(* IEC 61131-3 sources: brOscatLib/oscatBuild (part 2) *)

(* ---- oscatBuild.fun ---- *)
FUNCTION_BLOCK ACTUATOR_2P (* Actuators *)(* http://www.oscat.de/images/OSCATBuilding/oscat_building100_en.pdf#page=12 *)
    VAR_INPUT
        IN : BYTE;
        TEST : BOOL;
        ARE : BOOL := TRUE;
    END_VAR
    VAR_IN_OUT
        ARX : BOOL;
    END_VAR
    VAR_INPUT
        CYCLE_TIME : TIME;
        SENS : BYTE;
        SELF_ACT_TIME : TIME;
        SELF_ACT_PULSE : TIME;
        SELF_ACT_CYCLES : INT := 1;
    END_VAR
    VAR_OUTPUT
        OUT : BOOL;
        ARO : BOOL;
    END_VAR
    VAR
        timer : AUTORUN;
        pwgen : GEN_PULSE;
    END_VAR
END_FUNCTION_BLOCK
FUNCTION_BLOCK ACTUATOR_3P (* Actuators *)(* http://www.oscat.de/images/OSCATBuilding/oscat_building100_en.pdf#page=13 *)
    VAR_INPUT
        IN : BYTE;
        TEST : BOOL;
        ARE : BOOL := TRUE;
        END_POS : BOOL;
        T_RUN : TIME := TIME#1m0s0ms;
        T_EXT : TIME := TIME#10s0ms;
        T_CAL : TIME := TIME#10m0s0ms;
        T_DIAG : TIME := TIME#14400m0s0ms;
        SWITCH_AVAIL : BOOL;
    END_VAR
    VAR_IN_OUT
        ARX : BOOL;
    END_VAR
    VAR_OUTPUT
        OUT1 : BOOL;
        OUT2 : BOOL;
        POS : BYTE;
        ERROR : BOOL;
        STATUS : BYTE;
    END_VAR
    VAR
        ramp : _RMP_NEXT;
        tx : TIME;
        next_cal : TIME;
        next_diag : TIME;
        last : TIME;
        start : TIME;
    END_VAR
END_FUNCTION_BLOCK
FUNCTION_BLOCK ACTUATOR_A (* Actuators *)(* http://www.oscat.de/images/OSCATBuilding/oscat_building100_en.pdf#page=15 *)
    VAR_INPUT
        I1 : BYTE;
        IS : BOOL;
        I2 : BYTE;
        RV : BOOL;
        DX : BOOL;
        RUNTIME : TIME;
        SELF_ACT_TIME : TIME;
        OUT_MIN : WORD;
        OUT_MAX : WORD;
    END_VAR
    VAR_OUTPUT
        Y : WORD;
    END_VAR
    VAR
        timer : CYCLE_4;
        dx_edge : BOOL;
    END_VAR
END_FUNCTION_BLOCK
FUNCTION_BLOCK ACTUATOR_COIL (* Actuators *)(* http://www.oscat.de/images/OSCATBuilding/oscat_building100_en.pdf#page=16 *)
    VAR_INPUT
        IN : BOOL;
        SELF_ACT_CYCLE : TIME := TIME#14400m0s0ms;
        SELF_ACT_TIME : TIME := TIME#1s0ms;
    END_VAR
    VAR_OUTPUT
        OUT : BOOL;
        STATUS : BYTE;
    END_VAR
    VAR
        last : DWORD;
        init : BOOL;
        tx : DWORD;
        now : DWORD;
    END_VAR
END_FUNCTION_BLOCK
FUNCTION_BLOCK ACTUATOR_PUMP (* Actuators *)(* http://www.oscat.de/images/OSCATBuilding/oscat_building100_en.pdf#page=16 *)
    VAR_INPUT
        IN : BOOL;
        MANUAL : BOOL;
        RST : BOOL;
        MIN_ONTIME : TIME := TIME#10s0ms;
        MIN_OFFTIME : TIME := TIME#10s0ms;
        RUN_EVERY : TIME := TIME#10000m0s0ms;
    END_VAR
    VAR_OUTPUT
        PUMP : BOOL;
    END_VAR
    VAR_IN_OUT
        RUNTIME : UDINT;
        CYCLES : UDINT;
    END_VAR
    VAR
        tx : TIME;
        last_change : TIME;
        meter : ontime;
        old_man : BOOL;
        init : BOOL;
    END_VAR
END_FUNCTION_BLOCK
FUNCTION_BLOCK ACTUATOR_UD (* Actuators *)(* http://www.oscat.de/images/OSCATBuilding/oscat_building100_en.pdf#page=17 *)
    VAR_INPUT
        UD : BOOL;
        ON : BOOL;
        MANUAL : BOOL;
        UP : BOOL;
        DN : BOOL;
        OFF : BOOL;
        YUP_IN : BOOL;
        YDN_IN : BOOL;
        TON : TIME;
        TOFF : TIME;
        OUT_RETURN : BOOL;
    END_VAR
    VAR_OUTPUT
        YUP : BOOL;
        YDN : BOOL;
        STATUS : BYTE;
    END_VAR
    VAR
        tx : TIME;
        last : TIME;
        init : BOOL;
    END_VAR
END_FUNCTION_BLOCK
FUNCTION_BLOCK AUTORUN (* Actuators *)(* http://www.oscat.de/images/OSCATBuilding/oscat_building100_en.pdf#page=19 *)
    VAR_INPUT
        IN : BOOL;
        TEST : BOOL;
        ARE : BOOL := TRUE;
    END_VAR
    VAR_IN_OUT
        ARX : BOOL;
    END_VAR
    VAR_INPUT
        TRUN : TIME;
        TOFF : TIME;
    END_VAR
    VAR_OUTPUT
        OUT : BOOL;
        ARO : BOOL;
    END_VAR
    VAR
        timer : _RMP_B;
        val : BYTE;
    END_VAR
END_FUNCTION_BLOCK
FUNCTION_BLOCK CLICK (* Electrical *)(* http://www.oscat.de/images/OSCATBuilding/oscat_building100_en.pdf#page=47 *)
    VAR_INPUT
        IN : BOOL;
    END_VAR
    VAR_OUTPUT
        Q : BOOL;
        SINGLE : BOOL;
        DOUBLE : BOOL;
        TRIPLE : BOOL;
        STATUS : BYTE;
    END_VAR
    VAR_INPUT
        T_DEBOUNCE : TIME := TIME#10ms;
        T_SHORT : TIME := TIME#200ms;
        T_PAUSE : TIME := TIME#500ms;
        T_RECONFIG : TIME := TIME#1m0s0ms;
    END_VAR
    VAR
        s_in : SW_RECONFIG;
        tx : TIME;
        state : INT;
        last : TIME;
    END_VAR
END_FUNCTION_BLOCK
FUNCTION_BLOCK CLICK_MODE (* Electrical *)(* http://www.oscat.de/images/OSCATBuilding/oscat_building100_en.pdf#page=49 *)
    VAR_INPUT
        IN : BOOL;
    END_VAR
    VAR_OUTPUT
        SINGLE : BOOL;
        DOUBLE : BOOL;
        LONG : BOOL;
        TP_LONG : BOOL;
    END_VAR
    VAR_INPUT
        T_LONG : TIME := TIME#500ms;
    END_VAR
    VAR
        Timer : TP;
        cnt : INT;
        last : BOOL;
    END_VAR
END_FUNCTION_BLOCK
FUNCTION_BLOCK DEBOUNCE (* Electrical *)(* http://www.oscat.de/images/OSCATBuilding/oscat_building100_en.pdf#page=49 *)
    VAR_INPUT
        IN : BOOL;
        TD : TIME;
        PM : BOOL;
    END_VAR
    VAR_OUTPUT
        Q : BOOL;
    END_VAR
    VAR
        deb : TOF;
    END_VAR
END_FUNCTION_BLOCK
FUNCTION_BLOCK DIMM_2 (* Electrical *)(* http://www.oscat.de/images/OSCATBuilding/oscat_building100_en.pdf#page=50 *)
    VAR_INPUT
        SET : BOOL;
        VAL : BYTE := 255;
        I1 : BOOL;
        I2 : BOOL;
        RST : BOOL;
        T_DEBOUNCE : TIME := TIME#10ms;
        T_ON_MAX : TIME := TIME#0ms;
        T_DIMM_START : TIME := TIME#1s0ms;
        T_DIMM : TIME := TIME#3s0ms;
        MIN_ON : BYTE := 50;
        MAX_ON : BYTE := 255;
        RST_OUT : BOOL := TRUE;
        SOFT_DIMM : BOOL := TRUE;
        DBL1_TOG : BOOL;
        DBL2_TOG : BOOL;
        DBL1_SET : BOOL;
        DBL2_SET : BOOL;
        DBL1_POS : BYTE;
        DBL2_POS : BYTE;
    END_VAR
    VAR_OUTPUT
        Q : BOOL := FALSE;
        D1 : BOOL;
        D2 : BOOL;
    END_VAR
    VAR_IN_OUT
        OUT : BYTE;
    END_VAR
    VAR
        t1 : TOF;
        t2 : TOF;
        dc1 : CLICK_MODE;
        dc2 : CLICK_MODE;
        t3 : TON;
        dim : _RMP_B;
    END_VAR
END_FUNCTION_BLOCK
FUNCTION_BLOCK DIMM_I (* Electrical *)(* http://www.oscat.de/images/OSCATBuilding/oscat_building100_en.pdf#page=52 *)
    VAR_INPUT
        SET : BOOL;
        VAL : BYTE := 255;
        IN : BOOL;
        RST : BOOL;
        T_DEBOUNCE : TIME := TIME#10ms;
        T_RECONFIG : TIME := TIME#10s0ms;
        T_ON_MAX : TIME := TIME#0ms;
        T_DIMM_START : TIME := TIME#1s0ms;
        T_DIMM : TIME := TIME#3s0ms;
        MIN_ON : BYTE := 50;
        MAX_ON : BYTE := 255;
        SOFT_DIMM : BOOL := TRUE;
        DBL_TOGGLE : BOOL;
        RST_OUT : BOOL;
    END_VAR
    VAR_OUTPUT
        Q : BOOL := FALSE;
        DBL : BOOL;
    END_VAR
    VAR_IN_OUT
        OUT : BYTE;
    END_VAR
    VAR
        config : SW_RECONFIG;
        decode : CLICK_MODE;
        t3 : TON;
        dim : _RMP_B;
        dir : BOOL;
    END_VAR
END_FUNCTION_BLOCK
FUNCTION_BLOCK F_LAMP (* Electrical *)(* http://www.oscat.de/images/OSCATBuilding/oscat_building100_en.pdf#page=54 *)
    VAR_INPUT
        SWITCH : BOOL;
        DIMM : BYTE := 255;
        RST : BOOL;
    END_VAR
    VAR_OUTPUT
        LAMP : BYTE;
        STATUS : BYTE;
    END_VAR
    VAR_IN_OUT
        ONTIME : UDINT;
        CYCLES : UDINT;
    END_VAR
    VAR_INPUT
        T_NO_DIMM : UINT := 100;
        T_MAINTENANCE : UINT := 15000;
    END_VAR
    VAR
        runtime : ONTIME;
    END_VAR
END_FUNCTION_BLOCK
FUNCTION_BLOCK PULSE_LENGTH (* Electrical *)(* http://www.oscat.de/images/OSCATBuilding/oscat_building100_en.pdf#page=56 *)
    VAR_INPUT
        IN : BOOL;
    END_VAR
    VAR_OUTPUT
        SHORT : BOOL;
        MIDDLE : BOOL;
        LONG : BOOL;
    END_VAR
    VAR_INPUT
        T_SHORT : TIME := TIME#100ms;
        T_LONG : TIME := TIME#1s0ms;
    END_VAR
    VAR
        tx : TIME;
        tn : TIME;
        edge_ : BOOL;
    END_VAR
END_FUNCTION_BLOCK
FUNCTION_BLOCK PULSE_T (* Electrical *)(* http://www.oscat.de/images/OSCATBuilding/oscat_building100_en.pdf#page=56 *)
    VAR_INPUT
        IN : BOOL;
        T1 : TIME;
        T2 : TIME;
        RST : BOOL;
    END_VAR
    VAR_OUTPUT
        Q : BOOL;
    END_VAR
    VAR
        init : BOOL;
        last : TIME;
        tx : TIME;
        edge_ : BOOL;
    END_VAR
END_FUNCTION_BLOCK
FUNCTION_BLOCK SW_RECONFIG (* Electrical *)(* http://www.oscat.de/images/OSCATBuilding/oscat_building100_en.pdf#page=57 *)
    VAR_INPUT
        IN : BOOL;
        TD : TIME;
        TR : TIME;
    END_VAR
    VAR_OUTPUT
        Q : BOOL;
    END_VAR
    VAR
        T1 : TON;
        T2 : TON;
        INV : BOOL;
    END_VAR
END_FUNCTION_BLOCK
FUNCTION_BLOCK SWITCH_I (* Electrical *)(* http://www.oscat.de/images/OSCATBuilding/oscat_building100_en.pdf#page=58 *)
    VAR_INPUT
        SET : BOOL;
        IN : BOOL;
        RST : BOOL;
        T_DEBOUNCE : TIME := TIME#10ms;
        T_RECONFIG : TIME := TIME#1s0ms;
        T_ON_MAX : TIME := TIME#0ms;
    END_VAR
    VAR_OUTPUT
        Q : BOOL;
    END_VAR
    VAR
        state : BYTE;
        edge_ : BOOL;
        r_edge : BOOL;
        T_on : TIME;
        tx : TIME;
    END_VAR
END_FUNCTION_BLOCK
FUNCTION_BLOCK SWITCH_X (* Electrical *)(* http://www.oscat.de/images/OSCATBuilding/oscat_building100_en.pdf#page=59 *)
    VAR_INPUT
        IN1 : BOOL;
        IN2 : BOOL;
        IN3 : BOOL;
        IN4 : BOOL;
        IN5 : BOOL;
        IN6 : BOOL;
    END_VAR
    VAR_OUTPUT
        Q1 : BOOL;
        Q2 : BOOL;
        Q3 : BOOL;
        Q4 : BOOL;
        Q5 : BOOL;
        Q6 : BOOL;
        Q31 : BOOL;
        Q41 : BOOL;
        Q51 : BOOL;
        Q61 : BOOL;
        Q32 : BOOL;
        Q42 : BOOL;
        Q52 : BOOL;
        Q62 : BOOL;
    END_VAR
    VAR_INPUT
        T_DEBOUNCE : TIME := TIME#50ms;
    END_VAR
    VAR
        init : BOOL;
        T1 : TOF;
        T2 : TOF;
        T3 : TOF;
        T4 : TOF;
        T5 : TOF;
        T6 : TOF;
        tx : TIME;
        x1 : BOOL;
        x2 : BOOL;
        E1 : BOOL;
        E2 : BOOL;
    END_VAR
END_FUNCTION_BLOCK
FUNCTION_BLOCK TIMER_1 (* Electrical *)(* http://www.oscat.de/images/OSCATBasic/oscat_basic333_en.pdf#page=60 *)
    VAR_INPUT
        E : BOOL := TRUE;
        DTI : DT;
        START : TOD;
        DURATION : TIME;
        DAY : BYTE := 2#1111111;
    END_VAR
    VAR_OUTPUT
        Q : BOOL;
        STOP : TIME;
    END_VAR
END_FUNCTION_BLOCK
FUNCTION_BLOCK TIMER_2 (* Electrical *)(* http://www.oscat.de/images/OSCATBuilding/oscat_building100_en.pdf#page=60 *)
    VAR_INPUT
        DT_IN : DT;
        START : TOD;
        DURATION : TIME;
        MODE : BYTE;
        HOLIDAY : BOOL;
    END_VAR
    VAR_OUTPUT
        Q : BOOL;
    END_VAR
    VAR
        last_check : TIME;
        dat : DATE;
        daytime : TOD;
        activation : TIME;
        tx : TIME;
        enabled : BOOL;
        init : BOOL;
        wday : INT;
    END_VAR
    VAR RETAIN
        run_date : DATE;
    END_VAR
END_FUNCTION_BLOCK
FUNCTION TIMER_EVENT_DECODE : BOOL (* Electrical *)(* http://www.oscat.de/images/OSCATBuilding/oscat_building100_en.pdf#page=62 *)
    VAR_INPUT
        EVENT : STRING[STRING_LENGTH];
        LANG : INT;
    END_VAR
    VAR
        pos : INT;
        start : INT;
        stop : INT;
        pt : REFERENCE TO ARRAY[1..255] OF BYTE;
        step : INT;
        tmp : STRING[60];
    END_VAR
    VAR_IN_OUT
        RETVAL : TIMER_EVENT; (*Return value of the function*)
    END_VAR
END_FUNCTION
FUNCTION_BLOCK TIMER_EXT (* Electrical *)(* http://www.oscat.de/images/OSCATBuilding/oscat_building100_en.pdf#page=63 *)
    VAR_INPUT
        ENA : BOOL := TRUE;
        ON : BOOL;
        OFF : BOOL;
        MAN : BOOL;
        SWITCH : BOOL;
        DT_IN : DT;
        SUN_RISE : TOD;
        SUN_SET : TOD;
        HOLIDAY : BOOL;
        T_DEBOUNCE : TIME := TIME#100ms;
        T_RISE_START : TIME;
        T_RISE_STOP : TIME;
        T_SET_START : TIME;
        T_SET_STOP : TIME;
        T_DAY_START : TOD;
        T_DAY_STOP : TOD;
        ENABLE_SATURDAY : BOOL;
        ENABLE_SUNDAY : BOOL;
        ENABLE_HOLIDAY : BOOL;
    END_VAR
    VAR_OUTPUT
        Q : BOOL;
        STATUS : BYTE;
    END_VAR
    VAR
        mx : MANUAL_2;
        deb : DEBOUNCE;
        tdx : TOD;
        wdx : INT;
        tc : TIME;
        tx : DWORD;
        tl : DWORD;
        qx : BOOL;
        init : BOOL;
    END_VAR
END_FUNCTION_BLOCK
FUNCTION_BLOCK TIMER_P4 (* Electrical *)(* http://www.oscat.de/images/OSCATBuilding/oscat_building100_en.pdf#page=65 *)
    VAR_INPUT
        DTIME : DT;
        TREF_0 : TOD;
        TREF_1 : TOD;
        HOLY : BOOL;
        L0 : BOOL;
        L1 : BOOL;
        L2 : BOOL;
        L3 : BOOL;
        OFS : BYTE;
        ENQ : BOOL;
        MAN : BOOL;
        MI : BYTE;
        RST : BOOL;
    END_VAR
    VAR_IN_OUT
        PROG : ARRAY[0..array_max] OF TIMER_EVENT;
    END_VAR
    VAR_OUTPUT
        Q0 : BOOL;
        Q1 : BOOL;
        Q2 : BOOL;
        Q3 : BOOL;
        STATUS : BYTE;
    END_VAR
    VAR CONSTANT
        array_max : INT := 63;
        channel_max : INT := 3;
    END_VAR
    VAR
        day_start : DT;
        start : DT;
        event : TIMER_EVENT;
        pos : INT;
        last_execute : DT;
        current_day : DINT;
        mask : BYTE;
        ma : ARRAY[0..channel_max] OF BYTE;
        mo : ARRAY[0..channel_max] OF BYTE;
        qn : ARRAY[0..channel_max] OF BOOL;
        qs : ARRAY[0..channel_max] OF BOOL;
        channel : INT;
        tx : TOD;
    END_VAR
END_FUNCTION_BLOCK
FUNCTION AIR_DENSITY : REAL (* HLK *)(* http://www.oscat.de/images/OSCATBasic/oscat_basic333_en.pdf#page=426 *)
    VAR_INPUT
        T : REAL;
        P : REAL;
        RH : REAL;
    END_VAR
    VAR CONSTANT
        RL : REAL := 287.05;
        RX : REAL := 0.003773319;
    END_VAR
END_FUNCTION
FUNCTION AIR_ENTHALPY : REAL (* HLK *)(* http://www.oscat.de/images/OSCATBasic/oscat_basic333_en.pdf#page=427 *)
    VAR_INPUT
        T : REAL;
        RH : REAL;
    END_VAR
    VAR CONSTANT
        CPL : REAL := 1.00482;
        CW : REAL := 1.86;
        LH : REAL := 2500.78;
    END_VAR
END_FUNCTION
FUNCTION_BLOCK BOILER (* HLK *)(* http://www.oscat.de/images/OSCATBasic/oscat_basic333_en.pdf#page=428 *)
    VAR_INPUT
        T_UPPER : REAL;
        T_LOWER : REAL;
        PRESSURE : BOOL := TRUE;
        ENABLE : BOOL := TRUE;
        REQ_1 : BOOL;
        REQ_2 : BOOL;
        BOOST : BOOL;
        T_UPPER_MIN : REAL := 50;
        T_UPPER_MAX : REAL := 60;
        T_LOWER_ENABLE : BOOL;
        T_LOWER_MAX : REAL := 60;
        T_REQUEST_1 : REAL := 70;
        T_REQUEST_2 : REAL := 50;
        T_REQUEST_HYS : REAL := 5;
        T_PROTECT_HIGH : REAL := 80;
        T_PROTECT_LOW : REAL := 10;
    END_VAR
    VAR_OUTPUT
        HEAT : BOOL;
        ERROR : BOOL;
        STATUS : BYTE;
    END_VAR
    VAR
        edge_ : BOOL;
        boost_mode : BOOL;
        flag_0 : BOOL;
        flag_1 : BOOL;
        flag_2 : BOOL;
    END_VAR
END_FUNCTION_BLOCK
FUNCTION_BLOCK BURNER (* HLK *)(* http://www.oscat.de/images/OSCATBasic/oscat_basic333_en.pdf#page=430 *)
    VAR_INPUT
        IN : BOOL;
        STAGE2 : BOOL;
        OVER_TEMP : BOOL;
        OIL_TEMP : BOOL := TRUE;
        FLAME : BOOL;
        RST : BOOL;
        RST_TIMER : BOOL;
        PRE_HEAT_TIME : TIME := TIME#5s0ms;
        PRE_VENT_TIME : TIME := TIME#15s0ms;
        PRE_IGNITE_TIME : TIME := TIME#5s0ms;
        POST_IGNITE_TIME : TIME := TIME#25s0ms;
        STAGE2_DELAY : TIME := TIME#10s0ms;
        SAFETY_TIME : TIME := TIME#5s0ms;
        LOCKOUT_TIME : TIME := TIME#10s0ms;
        MULTIPLE_IGNITION : BOOL := TRUE;
        KW1 : REAL;
        KW2 : REAL;
    END_VAR
    VAR_OUTPUT
        MOTOR : BOOL;
        COIL1 : BOOL;
        COIL2 : BOOL;
        PRE_HEAT : BOOL;
        IGNITE : BOOL;
        KWH : REAL;
        STATUS : BYTE;
        FAIL : BOOL;
    END_VAR
    VAR_IN_OUT
        RUNTIME1 : UDINT;
        RUNTIME2 : UDINT;
        CYCLES : UDINT;
    END_VAR
    VAR
        state : BYTE;
        last : TIME;
        tx : TIME;
        last_change : TIME;
        timer1 : ONTIME;
        timer2 : ONTIME;
        oil_temp_last : BOOL;
        cycles2 : UDINT;
    END_VAR
END_FUNCTION_BLOCK
FUNCTION DEW_CON : REAL (* HLK *)(* http://www.oscat.de/images/OSCATBasic/oscat_basic333_en.pdf#page=434 *)
    VAR_INPUT
        RH : REAL;
        T : REAL;
    END_VAR
END_FUNCTION
FUNCTION DEW_RH : REAL (* HLK *)(* http://www.oscat.de/images/OSCATBasic/oscat_basic333_en.pdf#page=435 *)
    VAR_INPUT
        VC : REAL;
        T : REAL;
    END_VAR
END_FUNCTION
FUNCTION DEW_TEMP : REAL (* HLK *)(* http://www.oscat.de/images/OSCATBasic/oscat_basic333_en.pdf#page=436 *)
    VAR_INPUT
        RH : REAL;
        T : REAL;
    END_VAR
    VAR CONSTANT
        a : REAL := 7.5;
        b : REAL := 237.3;
    END_VAR
    VAR
        V : REAL;
    END_VAR
END_FUNCTION
FUNCTION HEAT_INDEX : REAL (* HLK *)(* http://www.oscat.de/images/OSCATBasic/oscat_basic333_en.pdf#page=436 *)
    VAR_INPUT
        T : REAL;
        RH : REAL;
    END_VAR
    VAR
        RH2 : REAL;
        T2 : REAL;
    END_VAR
END_FUNCTION
FUNCTION_BLOCK HEAT_METER (* HLK *)(* http://www.oscat.de/images/OSCATBasic/oscat_basic333_en.pdf#page=436 *)
    VAR_INPUT
        TF : REAL;
        TR : REAL;
        LPH : REAL;
        E : BOOL;
        RST : BOOL;
        CP : REAL;
        DENSITY : REAL;
        CONTENT : REAL;
        PULSE_MODE : BOOL;
        RETURN_METER : BOOL;
        AVG_TIME : TIME := TIME#5s0ms;
    END_VAR
    VAR_OUTPUT
        C : REAL;
    END_VAR
    VAR_IN_OUT
        Y : REAL;
    END_VAR
    VAR
        tx : DWORD;
        last : DWORD;
        int1 : FT_INT2;
        edge_ : BOOL;
        x : REAL;
        init : BOOL;
        y_last : REAL;
    END_VAR
END_FUNCTION_BLOCK
FUNCTION_BLOCK HEAT_TEMP (* HLK *)(* http://www.oscat.de/images/OSCATBasic/oscat_basic333_en.pdf#page=33 *)
    VAR_INPUT
        T_EXT : REAL;
        T_INT : REAL;
        OFFSET : REAL;
        T_REQ : REAL;
        TY_MAX : REAL := 70;
        TY_MIN : REAL := 25;
        TY_CONFIG : REAL := 70;
        T_INT_CONFIG : REAL := 20;
        T_EXT_CONFIG : REAL := -15;
        T_DIFF : REAL := 10;
        C : REAL := 1.33;
        H : REAL := 3;
    END_VAR
    VAR_OUTPUT
        TY : REAL;
        HEAT : BOOL;
    END_VAR
    VAR
        tr : REAL;
        tx : REAL;
    END_VAR
END_FUNCTION_BLOCK
FUNCTION_BLOCK LEGIONELLA (* HLK *)(* http://www.oscat.de/images/OSCATBasic/oscat_basic333_en.pdf#page=443 *)
    VAR_INPUT
        MANUAL : BOOL;
        TEMP_BOILER : REAL;
        TEMP_RETURN : REAL := 100;
        DT_IN : DT;
        RST : BOOL;
        T_START : TOD := TIME_OF_DAY#3:0;
        DAY : INT := 7;
        TEMP_SET : REAL := 70;
        TEMP_OFFSET : REAL := 10;
        TEMP_HYS : REAL := 5;
        T_MAX_HEAT : TIME := TIME#10m0s0ms;
        T_MAX_RET : TIME := TIME#10m0s0ms;
        TP_0 : TIME := TIME#5m0s0ms;
        TP_1 : TIME := TIME#5m0s0ms;
        TP_2 : TIME := TIME#5m0s0ms;
        TP_3 : TIME := TIME#5m0s0ms;
        TP_4 : TIME := TIME#5m0s0ms;
        TP_5 : TIME := TIME#5m0s0ms;
        TP_6 : TIME := TIME#5m0s0ms;
        TP_7 : TIME := TIME#5m0s0ms;
    END_VAR
    VAR_OUTPUT
        HEAT : BOOL;
        PUMP : BOOL;
        VALVE0 : BOOL;
        VALVE1 : BOOL;
        VALVE2 : BOOL;
        VALVE3 : BOOL;
        VALVE4 : BOOL;
        VALVE5 : BOOL;
        VALVE6 : BOOL;
        VALVE7 : BOOL;
        RUN : BOOL;
        STATUS : BYTE;
    END_VAR
    VAR
        X1 : TIMER_1;
        x2 : SEQUENCE_8;
        x3 : HYST_1;
        init : BOOL;
    END_VAR
END_FUNCTION_BLOCK
FUNCTION SDD : REAL (* HLK *)(* http://www.oscat.de/images/OSCATBasic/oscat_basic333_en.pdf#page=445 *)
    VAR_INPUT
        T : REAL;
        ICE : BOOL;
    END_VAR
END_FUNCTION
FUNCTION SDD_NH3 : REAL (* HLK *)(* http://www.oscat.de/images/OSCATBasic/oscat_basic333_en.pdf#page=446 *)
    VAR_INPUT
        T : REAL;
    END_VAR
END_FUNCTION
FUNCTION SDT_NH3 : REAL (* HLK *)(* http://www.oscat.de/images/OSCATBasic/oscat_basic333_en.pdf#page=446 *)
    VAR_INPUT
        P : REAL;
    END_VAR
END_FUNCTION
FUNCTION_BLOCK T_AVG24 (* HLK *)(* http://www.oscat.de/images/OSCATBasic/oscat_basic333_en.pdf#page=446 *)
    VAR_INPUT
        TS : INT;
        DTI : DT;
        RST : BOOL;
        T_FILTER : TIME := TIME#10m0s0ms;
        SCALE : REAL := 1;
        OFS : REAL;
    END_VAR
    VAR_OUTPUT
        TA : REAL;
        TP : BOOL;
    END_VAR
    VAR_IN_OUT
        T24 : REAL;
        T24_MAX : REAL;
        T24_MIN : REAL;
    END_VAR
    VAR
        samples : ARRAY[0..47] OF INT;
        pos : INT;
        init : BOOL;
        ft1 : FILTER_I;
        sum : DINT;
        last : DT;
    END_VAR
    VAR
        tmp_max : INT;
        tmp_min : INT;
        i : INT;
    END_VAR
END_FUNCTION_BLOCK
FUNCTION_BLOCK TANK_LEVEL (* HLK *)(* http://www.oscat.de/images/OSCATBuilding/oscat_building100_en.pdf#page=41 *)
    VAR_INPUT
        LEVEL : BOOL;
        LEAK : BOOL;
        ACLR : BOOL;
        MAX_VALVE_TIME : TIME;
        LEVEL_DELAY_TIME : TIME;
    END_VAR
    VAR_OUTPUT
        VALVE : BOOL;
        ALARM : BOOL;
        STATUS : BYTE;
    END_VAR
    VAR
        cx : ACTUATOR_COIL;
        tn : TON;
        tl : TONOF;
        open : BOOL;
    END_VAR
END_FUNCTION_BLOCK
FUNCTION TANK_VOL1 : REAL (* HLK *)(* http://www.oscat.de/images/OSCATBasic/oscat_basic333_en.pdf#page=448 *)
    VAR_INPUT
        TR : REAL;
        TL : REAL;
        H : REAL;
    END_VAR
END_FUNCTION
FUNCTION TANK_VOL2 : REAL (* HLK *)(* http://www.oscat.de/images/OSCATBasic/oscat_basic333_en.pdf#page=448 *)
    VAR_INPUT
        TR : REAL;
        H : REAL;
    END_VAR
END_FUNCTION
FUNCTION_BLOCK TEMP_EXT (* HLK *)(* http://www.oscat.de/images/OSCATBasic/oscat_basic333_en.pdf#page=449 *)
    VAR_INPUT
        T_EXT1 : REAL;
        T_EXT2 : REAL;
        T_EXT3 : REAL;
        T_EXT_CONFIG : BYTE;
        DT_IN : DT;
        T_EXT_MIN : REAL := -40;
        T_EXT_MAX : REAL := 60;
        T_EXT_DEFAULT : REAL := -10;
        HEAT_PERIOD_START : DATE := DATE#1970-9-1;
        HEAT_PERIOD_STOP : DATE := DATE#1970-4-30;
        COOL_PERIOD_START : DATE := DATE#1970-4-1;
        COOL_PERIOD_STOP : DATE := DATE#1970-9-30;
        HEAT_START_TEMP_DAY : REAL := 15;
        HEAT_START_TEMP_NIGHT : REAL := 10;
        HEAT_STOP_TEMP : REAL := 18;
        COOL_START_TEMP_DAY : REAL := 26;
        COOL_START_TEMP_NIGHT : REAL := 26;
        COOL_STOP_TEMP : REAL := 24;
        START_DAY : TOD := TIME_OF_DAY#9:0;
        START_NIGHT : TOD := TIME_OF_DAY#21:0;
        CYCLE_TIME : TIME := TIME#10m0s0ms;
    END_VAR
    VAR_OUTPUT
        T_EXT : REAL;
        HEAT : BOOL;
        COOL : BOOL;
    END_VAR
    VAR
        tx : TIME;
        last_run : TIME;
        init : BOOL;
        cool_start : DATE;
        cool_stop : DATE;
        heat_start : DATE;
        heat_stop : DATE;
        xdate : DATE;
        day : BOOL;
    END_VAR
END_FUNCTION_BLOCK
FUNCTION WATER_CP : REAL (* HLK *)(* http://www.oscat.de/images/OSCATBasic/oscat_basic333_en.pdf#page=452 *)
    VAR_INPUT
        T : REAL;
    END_VAR
    VAR
        Pts : INT := 10;
        data : ARRAY[1..20, 0..1] OF REAL := [0, 4.228, 5, 4.2, 10, 4.188, 15, 4.184, 50, 4.181, 60, 4.183, 70, 4.187, 80, 4.194, 90, 4.204, 100, 4.22];
    END_VAR
END_FUNCTION
FUNCTION WATER_DENSITY : REAL (* HLK *)(* http://www.oscat.de/images/OSCATBasic/oscat_basic333_en.pdf#page=452 *)
    VAR_INPUT
        T : REAL;
        SAT : BOOL;
    END_VAR
    VAR CONSTANT
        a0 : REAL := 999.83952;
        a1 : REAL := 16.952577;
        a2 : REAL := -0.0079905127;
        a3 : REAL := -4.6241757E-05;
        a4 : REAL := 1.0584601E-07;
        a5 : REAL := -2.8103006E-10;
        b : REAL := 0.0168872;
    END_VAR
    VAR
        T2 : REAL;
        T4 : REAL;
    END_VAR
END_FUNCTION
FUNCTION WATER_ENTHALPY : REAL (* HLK *)(* http://www.oscat.de/images/OSCATBasic/oscat_basic333_en.pdf#page=453 *)
    VAR_INPUT
        T : REAL;
    END_VAR
    VAR
        Pts : INT := 11;
        data : ARRAY[1..20, 0..1] OF REAL := [0, 0.06, 10, 42.1, 20, 83.9, 30, 125.8, 40, 167.58, 50, 209.4, 60, 251.2, 70, 293.1, 80, 335, 90, 377, 100, 419.1];
    END_VAR
END_FUNCTION
FUNCTION WCT : REAL (* HLK *)(* http://www.oscat.de/images/OSCATBasic/oscat_basic333_en.pdf#page=453 *)
    VAR_INPUT
        T : REAL;
        V : REAL;
    END_VAR
END_FUNCTION
FUNCTION_BLOCK BLIND_ACTUATOR (* Jalousie *)(* http://www.oscat.de/images/OSCATBuilding/oscat_building100_en.pdf#page=74 *)
    VAR_INPUT
        UP : BOOL;
        DN : BOOL;
        S_IN : BYTE;
        T_UD : TIME := TIME#10s0ms;
        T_ANGLE : TIME := TIME#3s0ms;
        T_LOCKOUT : TIME := TIME#100ms;
    END_VAR
    VAR_OUTPUT
        POS : BYTE;
        ANG : BYTE;
        QU : BOOL;
        QD : BOOL;
        STATUS : BYTE;
    END_VAR
    VAR
        position : RMP_B;
        angle : RMP_B;
        lock : INTERLOCK;
    END_VAR
END_FUNCTION_BLOCK
FUNCTION_BLOCK BLIND_CONTROL (* Jalousie *)(* http://www.oscat.de/images/OSCATBuilding/oscat_building100_en.pdf#page=75 *)
    VAR_INPUT
        UP : BOOL;
        DN : BOOL;
        S_IN : BYTE;
        PI : BYTE;
        AI : BYTE;
        T_UD : TIME;
        T_ANGLE : TIME;
        SENS : BYTE := 5;
        T_LOCKOUT : TIME := TIME#100ms;
    END_VAR
    VAR_OUTPUT
        POS : BYTE;
        ANG : BYTE;
        MU : BOOL;
        MD : BOOL;
        STATUS : BYTE;
    END_VAR
    VAR
        act : BLIND_ACTUATOR;
        delta : BYTE;
        bTimeTest : BOOL := FALSE;
        iPos : BYTE;
        iAngel : BYTE;
    END_VAR
END_FUNCTION_BLOCK
FUNCTION_BLOCK BLIND_CONTROL_S (* Jalousie *)(* http://www.oscat.de/images/OSCATBuilding/oscat_building100_en.pdf#page=78 *)
    VAR_INPUT
        UP : BOOL;
        DN : BOOL;
        S_IN : BYTE := 125;
        PI : BYTE;
        T_UP : TIME;
        T_DN : TIME;
        RU : BOOL;
        RD : BOOL;
        T_LOCKOUT : TIME := TIME#100ms;
        T_EXT : TIME;
        EXT_TRIG : BYTE := 5;
        R_POS_TOP : BYTE := 255;
        R_POS_BOT : BYTE;
    END_VAR
    VAR_OUTPUT
        POS : BYTE;
        MU : BOOL;
        MD : BOOL;
        STATUS : BYTE;
    END_VAR
    VAR
        rmp : _RMP_NEXT;
        tx : TIME;
        last : TIME;
        PI_last : BYTE;
    END_VAR
END_FUNCTION_BLOCK
FUNCTION_BLOCK BLIND_INPUT (* Jalousie *)(* http://www.oscat.de/images/OSCATBuilding/oscat_building100_en.pdf#page=80 *)
    VAR_INPUT
        POS : BYTE;
        ANG : BYTE;
        S1 : BOOL;
        S2 : BOOL;
        IN : BOOL;
        PI : BYTE;
        AI : BYTE;
        SINGLE_SWITCH : BOOL;
        CLICK_EN : BOOL := TRUE;
        CLICK_TIME : TIME := TIME#500ms;
        MAX_RUNTIME : TIME := TIME#1m0s0ms;
        MANUAL_TIMEOUT : TIME := TIME#60m0s0ms;
        DEBOUNCE_TIME : TIME := TIME#20ms;
        DBL_CLK1 : BOOL := FALSE;
        DBL_POS1 : BYTE;
        DBL_ANG1 : BYTE;
        DBL_CLK2 : BOOL := FALSE;
        DBL_POS2 : BYTE := 255;
        DBL_ANG2 : BYTE := 255;
        D1_TOGGLE : BOOL := TRUE;
        D2_TOGGLE : BOOL := TRUE;
        MASTER_MODE : BOOL;
    END_VAR
    VAR_OUTPUT
        QU : BOOL := TRUE;
        QD : BOOL := TRUE;
        STATUS : BYTE;
        PO : BYTE := 255;
        AO : BYTE := 255;
        D1 : BOOL;
        D2 : BOOL;
    END_VAR
    VAR
        s1e : TOF;
        s2e : TOF;
        s1d : CLICK_MODE;
        s2d : CLICK_MODE;
        dir : BOOL;
        tx : TIME;
        last : TIME;
    END_VAR
END_FUNCTION_BLOCK
FUNCTION_BLOCK BLIND_NIGHT (* Jalousie *)(* http://www.oscat.de/images/OSCATBuilding/oscat_building100_en.pdf#page=84 *)
    VAR_INPUT
        UP : BOOL;
        DN : BOOL;
        S_IN : BYTE;
        PI : BYTE;
        AI : BYTE;
        E_NIGHT : BOOL := TRUE;
        E_DAY : BOOL := TRUE;
        DTIN : DT;
        SUNRISE : TOD;
        SUNSET : TOD;
        SUNRISE_OFFSET : TIME;
        SUNSET_OFFSET : TIME;
        NIGHT_POSITION : BYTE;
        NIGHT_ANGLE : BYTE;
    END_VAR
    VAR_OUTPUT
        QU : BOOL;
        QD : BOOL;
        STATUS : BYTE;
        PO : BYTE;
        AO : BYTE;
    END_VAR
    VAR
        night : BOOL;
        last_night : DATE;
        last_day : DATE;
    END_VAR
END_FUNCTION_BLOCK
FUNCTION_BLOCK BLIND_SCENE (* Jalousie *)(* http://www.oscat.de/images/OSCATBuilding/oscat_building100_en.pdf#page=87 *)
    VAR_INPUT
        UP : BOOL;
        DN : BOOL;
        S_IN : BYTE;
        PI : BYTE;
        AI : BYTE;
        ENABLE : BOOL;
        SWRITE : BOOL;
        SCENE : BYTE;
    END_VAR
    VAR_OUTPUT
        QU : BOOL;
        QD : BOOL;
        STATUS : BYTE;
        PO : BYTE;
        AO : BYTE;
    END_VAR
    VAR RETAIN
        sx : ARRAY[0..15, 0..2] OF BYTE;
    END_VAR
    VAR
        x : BYTE;
    END_VAR
END_FUNCTION_BLOCK
FUNCTION_BLOCK BLIND_SECURITY (* Jalousie *)(* http://www.oscat.de/images/OSCATBuilding/oscat_building100_en.pdf#page=89 *)
    VAR_INPUT
        UP : BOOL;
        DN : BOOL;
        S_IN : BYTE;
        PI : BYTE;
        AI : BYTE;
        FIRE : BOOL;
        WIND : BOOL;
        ALARM : BOOL;
        DOOR : BOOL;
        RAIN : BOOL;
        ALARM_UP : BOOL := TRUE;
        WIND_UP : BOOL := TRUE;
        RAIN_UP : BOOL := FALSE;
    END_VAR
    VAR_OUTPUT
        QU : BOOL;
        QD : BOOL;
        STATUS : BYTE;
        PO : BYTE;
        AO : BYTE;
    END_VAR
END_FUNCTION_BLOCK
FUNCTION_BLOCK BLIND_SET (* Jalousie *)(* http://www.oscat.de/images/OSCATBuilding/oscat_building100_en.pdf#page=91 *)
    VAR_INPUT
        UP : BOOL;
        DN : BOOL;
        S_IN : BYTE;
        PI : BYTE;
        AI : BYTE;
        IN : BOOL;
        PX : BYTE;
        AX : BYTE;
        OVERRIDE_MANUAL : BOOL;
        RESTORE_POSITION : BOOL;
        RESTORE_TIME : TIME := TIME#1m0s0ms;
    END_VAR
    VAR_OUTPUT
        QU : BOOL;
        QD : BOOL;
        STATUS : BYTE;
        PO : BYTE;
        AO : BYTE;
    END_VAR
    VAR
        tx : TIME;
        ps : BYTE;
        as : BYTE;
        last : TIME;
    END_VAR
END_FUNCTION_BLOCK
FUNCTION_BLOCK BLIND_SHADE (* Jalousie *)(* http://www.oscat.de/images/OSCATBuilding/oscat_building100_en.pdf#page=93 *)
    VAR_INPUT
        UP : BOOL;
        DN : BOOL;
        S_IN : BYTE;
        PI : BYTE;
        AI : BYTE;
        ENABLE : BOOL;
        SUN : BOOL;
    END_VAR
    VAR_IN_OUT
        CX : CALENDAR;
    END_VAR
    VAR_INPUT
        SUNRISE_OFFSET : TIME := TIME#60m0s0ms;
        SUNSET_PRESET : TIME := TIME#60m0s0ms;
        DIRECTION : REAL := 180;
        ANGLE_OFFSET : REAL := 80;
        SLAT_WIDTH : REAL := 80;
        SLAT_SPACING : REAL := 60;
        SHADE_DELAY : TIME := TIME#1m0s0ms;
        SHADE_POS : BYTE;
    END_VAR
    VAR_OUTPUT
        QU : BOOL;
        QD : BOOL;
        STATUS : BYTE;
        PO : BYTE;
        AO : BYTE;
    END_VAR
    VAR
        angle : REAL;
        sun_delay : TOF;
    END_VAR
END_FUNCTION_BLOCK
FUNCTION_BLOCK BLIND_SHADE_S (* Jalousie *)(* http://www.oscat.de/images/OSCATBuilding/oscat_building100_en.pdf#page=96 *)
    VAR_INPUT
        UP : BOOL;
        DN : BOOL;
        S_IN : BYTE;
        PI : BYTE;
        ENABLE : BOOL;
        SUN : BOOL;
        HORZ1 : REAL := 100;
        HORZ2 : REAL := 260;
        VERT : REAL := 90;
        ALERT : BOOL := FALSE;
    END_VAR
    VAR_IN_OUT
        CX : calendar;
    END_VAR
    VAR_INPUT
        SUNRISE_OFFSET : TIME := TIME#60m0s0ms;
        SUNSET_PRESET : TIME := TIME#60m0s0ms;
        SHADE_DELAY : TIME := TIME#1m0s0ms;
        SHADE_POS : BYTE;
    END_VAR
    VAR_OUTPUT
        QU : BOOL;
        QD : BOOL;
        STATUS : BYTE;
        PO : BYTE;
    END_VAR
    VAR
        sun_delay : TOF;
    END_VAR
END_FUNCTION_BLOCK
FUNCTION BUILDING_VERSION : DWORD (* Other *)(* http://www.oscat.de/images/OSCATBuilding/oscat_building100_en.pdf#page=11 *)
    VAR_INPUT
        IN : BOOL;
    END_VAR
END_FUNCTION

(* ---- PULSE_LENGTH.st ---- *)
FUNCTION_BLOCK PULSE_LENGTH
    (*http://www.oscat.de/images/OSCATBuilding/oscat_building100_en.pdf#page=56*)
    (* read system time *)
    tx := DWORD_TO_TIME(T_PLC_MS());

    (* reset outputs, they should only be active 1 cycle *)
    SHORT := FALSE;
    MIDDLE := FALSE;
    LONG := FALSE;

    (* detect rising edge_ *)
    IF IN AND NOT edge_ THEN
    	edge_ := TRUE;
    	tn := tx;

    (* detect for falling edge_ *)
    ELSIF NOT IN AND edge_ THEN
    	edge_ := FALSE;
    	tn := tx - tn;
    	IF tn < T_SHORT THEN
    		SHORT := TRUE;
    	ELSIF tn > T_LONG THEN
    		LONG := TRUE;
    	ELSE
    		MIDDLE := TRUE;
    	END_IF

    (* generate LONG pulse as soon as T_LONG is reached *)
    ELSIF IN AND tx - tn > T_LONG THEN
    	LONG := TRUE;
    END_IF

    (* revision history

    hm	15. feb 2006	rev 1.0
    	original version

    hm	15 sep 2007		rev 1.1
    	replaced Time() with T_PLC_MS for compatibility and performance reasons

    *)
END_FUNCTION_BLOCK

(* ---- PULSE_T.st ---- *)
FUNCTION_BLOCK PULSE_T
    (*http://www.oscat.de/images/OSCATBuilding/oscat_building100_en.pdf#page=56*)
    tx := DWORD_TO_TIME(T_PLC_MS());
    IF NOT init THEN
    	init := TRUE;
    	last := tx;
    ELSIF RST THEN
    	(* asynchronous reset *)
    	Q := FALSE;
    ELSIF IN AND NOT edge_ AND NOT Q THEN
    	(* a rising edge_ on IN will reversre the output status, if new pulse is startet the start time is stored IN last *)
    	last := tx;
    	Q := TRUE;
    ELSIF NOT IN AND edge_ AND ((tx - last) > T1) THEN
    	(* a falling edge_ on IN will clear the output if IN was high for more then T1 *)
    	Q := FALSE;
    ELSIF (tx - last) >= T2 THEN
    	(* timeout for long pulse if second click did not occur or IN stays high *)
    	Q := FALSE;
    END_IF

    edge_ := IN;

    (* revision histroy
    hm	15. jul. 2008	rev 1.0
    	original release

    *)

END_FUNCTION_BLOCK

(* ---- SW_RECONFIG.st ---- *)
FUNCTION_BLOCK SW_RECONFIG
    (*http://www.oscat.de/images/OSCATBuilding/oscat_building100_en.pdf#page=57*)
    (* run debounce circuit *)
    T1(IN := IN, PT := TD);

    IF TR > t#0s THEN
    	(* generate output *)
    	Q := T1.Q XOR INV;
    	(* reconfiguration timer *)
    	T2(IN := Q, pt := TR);
    	(* when T2.Q goes high then reverse INV *)
    	IF T2.Q THEN INV := NOT INV; END_IF
    ELSE
    	Q := T1.Q;
    END_IF

    (* revision history
    hm	22.10.2008	rev 1.0
    	original version

    *)

END_FUNCTION_BLOCK

(* ---- SWITCH_I.st ---- *)
FUNCTION_BLOCK SWITCH_I
    (*http://www.oscat.de/images/OSCATBuilding/oscat_building100_en.pdf#page=58*)
    (* read system time *)
    tx := DWORD_TO_TIME(T_PLC_MS());

    (* asynchronous SET and reset first *)
    IF SET AND NOT RST THEN
    	Q := TRUE;
    	T_on := tx;
    ELSIF RST THEN
    	Q := FALSE;
    (* check FOR input edge_ AND start debounce timer *)
    ELSIF (IN XOR edge_) AND NOT (state = 1) THEN
    	state := 1;
    	T_on := tx;
    (* edge_ was detected and debounce time elapsed *)
    ELSIF (state = 1) AND (tx - T_DEBOUNCE >= T_on) THEN
    	state := 2;
    	(* react on rising or falling edge_ depending on r_edge *)
    	IF r_edge XOR IN THEN Q := NOT Q; END_IF
    (* wait for T_RECONFIG and adjust r_edge *)
    ELSIF state = 2 AND tx - T_RECONFIG >= T_on THEN
    	r_edge := IN;
    END_IF
    IF Q AND T_ON_MAX > t#0ms AND tx >= T_on + T_ON_MAX THEN
    	Q := FALSE;
    END_IF
    edge_ := IN;

    (* revision history

    hm	4 aug 2006	rev 1.0
    	original version

    hm	15.9.2007	rev 1.1
    	replaced Time() with T_PLC_MS for compatibility and performance reasons

    *)
END_FUNCTION_BLOCK

(* ---- SWITCH_X.st ---- *)
FUNCTION_BLOCK SWITCH_X
    (*http://www.oscat.de/images/OSCATBuilding/oscat_building100_en.pdf#page=59*)
    (* initialize on startup *)
    IF NOT init THEN
    	init := TRUE;
    	IF T_DEBOUNCE < t#50ms THEN tx := t#50ms; ELSE tx := T_DEBOUNCE; END_IF
    	T1(PT := tx);
    	T2(PT := tx);
    	T3(PT := tx);
    	T4(PT := tx);
    	T5(PT := tx);
    	T6(PT := tx);
    ELSE
    	Q1 := FALSE;
    	Q2 := FALSE;
    	Q3 := FALSE;
    	Q4 := FALSE;
    	Q5 := FALSE;
    	Q6 := FALSE;
    	Q31 := FALSE;
    	Q41 := FALSE;
    	Q51 := FALSE;
    	Q61 := FALSE;
    	Q32 := FALSE;
    	Q42 := FALSE;
    	Q52 := FALSE;
    	Q62 := FALSE;
    END_IF

    (* read inputs and debounce *)
    	T1(IN := IN1);
    	T2(IN := IN2);
    	T3(IN := IN3);
    	T4(IN := IN4);
    	T5(IN := IN5);
    	T6(IN := IN6);

    (* detect edge of IN1 and IN2 *)
    IF T1.Q AND NOT E1 THEN x1 := TRUE; END_IF
    IF T2.Q AND NOT E2 THEN x2 := TRUE; END_IF

    IF T1.Q THEN
    	IF T3.q THEN
    		Q31 := TRUE;
    		x1 := FALSE;
    	ELSIF T4.q THEN
    		Q41 := TRUE;
    		x1 := FALSE;
    	ELSIF T5.q THEN
    		Q51 := TRUE;
    		x1 := FALSE;
    	ELSIF T6.q THEN
    		Q61 := TRUE;
    		x1 := FALSE;
    	END_IF
    ELSIF T2.Q THEN
    	IF T3.q THEN
    		Q32 := TRUE;
    		x2 := FALSE;
    	ELSIF T4.q THEN
    		Q42 := TRUE;
    		x2 := FALSE;
    	ELSIF T5.q THEN
    		Q52 := TRUE;
    		x2 := FALSE;
    	ELSIF T6.q THEN
    		Q62 := TRUE;
    		x2 := FALSE;
    	END_IF
    (* IN1 was active alone *)
    ELSIF NOT T1.Q AND E1 AND x1 THEN
    	Q1 := TRUE;
    	x1 := FALSE;
    ELSIF NOT T2.Q AND E2 AND x2 THEN
    	Q2 := TRUE;
    	x2 := FALSE;
    ELSIF T3.Q THEN
    	Q3 := TRUE;
    ELSIF T4.Q THEN
    	Q4 := TRUE;
    ELSIF T5.Q THEN
    	Q5 := TRUE;
    ELSIF T6.Q THEN
    	Q6 := TRUE;
    END_IF

    (* save state of IN1 and IN2 *)
    E1 := T1.Q;
    E2 := T2.Q;

END_FUNCTION_BLOCK

(* ---- T_AVG24.st ---- *)
FUNCTION_BLOCK T_AVG24
    (*http://www.oscat.de/images/OSCATBasic/oscat_basic333_en.pdf#page=446*)
    (* first filter the sensor readings *)
    ft1(X := TS, T := T_FILTER);

    IF RST OR NOT init THEN
    	init := TRUE;
    	IF T24 = -1000.0 THEN T24 := INT_TO_REAL(ft1.Y) * 0.1; END_IF
    	FOR pos := 0 TO 47 DO
    		samples[pos] := REAL_TO_INT(T24 * 10.0);
    	END_FOR
    	pos := 0;
    	sum := INT_TO_DINT(samples[0]) * 48;
    	(* calculate the output value *)
    	TA := (INT_TO_REAL(ft1.Y) * 0.1 + OFS) * SCALE;
    	T24 := (DINT_TO_REAL(sum) * 0.00208333333333 + OFS) * SCALE;
    	TP := TRUE;
    ELSIF DT_TO_DWORD(DTI) / 60 MOD 30 = 0 AND DTI > last THEN
    	(* make sure we onlyexecute once every 30 mins *)
    	last := DTI + T#1m;
    	(* sample the temperature every 30 mins and store in ring buffer samples *)
    	(* sum always holds the sum of the array *)
    	(* subtract the oldest sample from sum *)
    	sum := sum - INT_TO_DINT(samples[pos]);
    	(* strore the new sample *)
    	samples[pos] := ft1.Y;
    	(* add the new sample to sum *)
    	sum := sum + INT_TO_DINT(samples[pos]);
    	(* increment the counter for the next sample *)
    	pos := INC1(pos, 48);
    	(* calculate the output value *)
    	TA := (INT_TO_REAL(ft1.Y) * 0.1 + OFS) * SCALE;
    	T24 := (DINT_TO_REAL(sum) * 0.00208333333333 + OFS) * SCALE;
    	(* calculate the min and max over the last 24 hours *)
    	tmp_max := -32000;
    	tmp_min := 32000;
    	FOR i := 0 TO 47 DO
    		tmp_max := MAX(tmp_max, samples[i]);
    		tmp_min := MIN(tmp_min, samples[i]);
    	END_FOR
    	T24_MAX := (INT_TO_REAL(tmp_max) * 0.1 + OFS) * SCALE;
    	T24_MIN := (INT_TO_REAL(tmp_min) * 0.1 + OFS) * SCALE;
    	TP := TRUE;
    ELSE
    	TP := FALSE;
    END_IF

    (* revision history
    hm	3. nov. 2008	rev 1.0
    	original version

    hm	8. feb. 2009	rev 1.1
    	changes sign of OFS
    	added outputs T24_MIN and T24_MAX

    hm	13. mar. 2009	rev 1.2
    	improved code
    *)
END_FUNCTION_BLOCK

(* ---- TANK_LEVEL.st ---- *)
FUNCTION_BLOCK TANK_LEVEL
    (*http://www.oscat.de/images/OSCATBuilding/oscat_building100_en.pdf#page=41*)
    (* preprocess the LEVEL information *)
    tl(in := LEVEL, T_ON := LEVEL_DELAY_TIME, T_OFF := LEVEL_DELAY_TIME);
    open := tl.Q;

    (* start logic *)
    IF ALARM THEN
    	(* check for ACLR if ALARM is present *)
    	IF ACLR THEN
    		ALARM := FALSE;
    		STATUS := 101; (* ACLR pressed *)
    		cx(in := FALSE);
    	END_IF
    	RETURN;
    ELSIF LEAK THEN
    	(* leakeage detected *)
    	cx(in := FALSE);
    	ALARM := TRUE;
    	STATUS := 1;	(* leakeage error *)
    ELSIF open THEN
    	(* VALVE needs to be opened because LEVEL is too low *)
    	cx(in := TRUE);
    	STATUS := 102; (* VALVE open by low LEVEL *)
    ELSE
    	(* VALVE needs to be closed *)
    	cx(in := FALSE);
    	STATUS := 100; (* VALVE idle *)
    END_IF

    (* check if VALVE is open too long and generate ALARM if necessary *)
    tn(in := cx.out AND (MAX_VALVE_TIME > T#0s), PT := MAX_VALVE_TIME);
    IF tn.Q THEN
    	ALARM := TRUE;
    	STATUS := 2; (* overtime error *)
    	cx(in := FALSE);
    END_IF

    (* set output signal *)
    VALVE := cx.out;

    (* revision history
    hm 27. feb 2007	rev 1.0
    	original version

    hm	24. jul 2009	rev 1.1
    	changed parameters of tonof

    *)
END_FUNCTION_BLOCK

(* ---- TEMP_EXT.st ---- *)
FUNCTION_BLOCK TEMP_EXT
    (*http://www.oscat.de/images/OSCATBasic/oscat_basic333_en.pdf#page=449*)
    IF NOT init THEN
    	init := TRUE;
    	heat_start := SET_DATE(1972,MONTH_OF_DATE(HEAT_PERIOD_START),DAY_OF_MONTH(HEAT_PERIOD_START));
    	heat_stop := SET_DATE(1972,MONTH_OF_DATE(HEAT_PERIOD_STOP),DAY_OF_MONTH(HEAT_PERIOD_STOP));
    	cool_start := SET_DATE(1972,MONTH_OF_DATE(COOL_PERIOD_START),DAY_OF_MONTH(COOL_PERIOD_START));
    	cool_stop := SET_DATE(1972,MONTH_OF_DATE(COOL_PERIOD_STOP),DAY_OF_MONTH(COOL_PERIOD_STOP));
    END_IF

    (* read system time *)
    tx := DWORD_TO_TIME(T_PLC_MS());

    (* for efficiency exit isf this program has been executed less then 1min ago *)
    IF tx - last_run < CYCLE_TIME THEN RETURN; END_IF

    (* calculate frequently used variables *)
    xdate := SET_DATE(1972,MONTH_OF_DATE(DT_TO_DATE(DT_IN)),DAY_OF_MONTH(DT_TO_DATE(DT_IN)));
    day := DT_TO_TOD(DT_IN) >= START_DAY AND  DT_TO_TOD(DT_IN) < START_NIGHT;

    (* read the correct external temperature depending on the T_EXT_CONFIG setting *)
    T_EXT := MULTI_IN(T_EXT1, T_EXT2, T_EXT3, T_EXT_DEFAULT, T_EXT_MIN, T_EXT_MAX, T_EXT_CONFIG);

    (* dtermine heating *)
    IF (heat_start <= heat_stop AND xdate >= heat_start AND xdate <= heat_stop) OR (heat_start > heat_stop AND (xdate >= heat_start OR xdate <= heat_stop)) THEN
    	(* heating period id true check for temperature *)
    	IF day AND T_EXT <= HEAT_START_TEMP_DAY THEN
    		HEAT := TRUE;
    	ELSIF NOT day AND T_EXT <= HEAT_START_TEMP_NIGHT THEN
    		HEAT := TRUE;
    	ELSIF T_EXT >= HEAT_STOP_TEMP THEN
    		HEAT := FALSE;
    	END_IF
    ELSE
    	HEAT := FALSE;
    END_IF

    (* dtermine cooling *)
    IF (cool_start <= cool_stop AND xdate >= cool_start AND xdate <= cool_stop) OR (cool_start > cool_stop AND (xdate >= cool_start OR xdate <= cool_stop)) THEN
    	(* cooling period is true check for temperature *)
    	IF day AND T_EXT >= COOL_START_TEMP_DAY THEN
    		COOL := TRUE;
    	ELSIF NOT day AND T_EXT >= COOL_START_TEMP_NIGHT THEN
    		COOL := TRUE;
    	ELSIF T_EXT <= COOL_STOP_TEMP THEN
    		COOL := FALSE;
    	END_IF
    ELSE
    	COOL := FALSE;
    END_IF

    last_run := tx;

    (* revision history
    hm	6 dec 2006	rev 1.0
    	original version

    hm	15.9.2007		rev 1.1
    	replaced Time() with T_PLC_MS for compatibility and performance reasons

    hm	7. oct. 2008	rev 1.2
    	changed name of function month to month_of_date

    hm	13. mar. 2009	rev 1.3
    	real constants updated to new systax using dot

    *)

END_FUNCTION_BLOCK

(* ---- TIMER_1.st ---- *)
FUNCTION_BLOCK TIMER_1
    (*http://www.oscat.de/images/OSCATBasic/oscat_basic333_en.pdf#page=60*)
    IF E THEN
    	STOP := TOD_TO_TIME(START) + DURATION;
    	IF STOP > T#24h THEN STOP := STOP - T#24h; END_IF
    	Q := TIMECHECK(DT_TO_TOD(DTI), START, TIME_TO_TOD(STOP)) AND (SHR(BYTE#128, DAY_OF_WEEK(DT_TO_DATE(DTI))) AND DAY) > BYTE#0;
    ELSE
    	Q := FALSE; (* clear output when E is not true *)
    END_IF

    (*
    1.12.2006 hm		rev 1.1
    	corrected an error with pulse width = 0.

    25.12.2006 hm		rev 1.2
    	corrected an error when timer overflows.

    14.apr 2007 hm		rev 1.3
    	corrected an error while while output would not go active when START year would be 1970.
    	increase accuracy by checking every 100ms
    	added init section to compensate for timer overflow

    15.9.2007 hm		rev 1.4
    	replaced Time() with T_PLC_MS for compatibility and performance reasons

    hm	1. okt 2007		rev 1.5
    	corrected an error while output would not stay active over midnight.

    hm	17. jan 2008	rev 1.6
    	New code with better performance
    	Output is now only active during the time of DAY it is supposed to
    	no pulse is generated at power up

    hm	7. oct. 2008	rev 1.7
    	changed function weekday to day_of_week

    hm	23. oct. 2008	rev 2.0
    	new code, added input E, now days can be selected by bits in byte DAY

    hm	6. nov. 2008	rev 2.1
    	added default for input EN and input DAY

    hm 16. dec 2009	rev 2.2
    	fixed a bug over midnight

    *)
END_FUNCTION_BLOCK

(* ---- TIMER_2.st ---- *)
FUNCTION_BLOCK TIMER_2
    (*http://www.oscat.de/images/OSCATBuilding/oscat_building100_en.pdf#page=60*)
    (* read system time *)
    tx := DWORD_TO_TIME(T_PLC_MS());

    IF NOT init THEN
    	init := TRUE;
    	last_check := tx - t#100ms;
    END_IF

    (* for performance resons exit if execution is not necessary *)
    IF tx - last_check < T#100ms THEN RETURN; END_IF

    (* calculate temp variables *)
    dat := DT_TO_DATE(DT_IN);
    daytime := DT_TO_TOD(DT_IN);
    wday := DAY_OF_WEEK(dat);

    (* calculate if any action is necessary today *)
    CASE MODE OF
    	1..7:	(* mondays to fridays *)
    		enabled := wday = BYTE_TO_INT(MODE);
    	11:	(* every day *)
    		enabled := TRUE;
    	12..16:	(* every nth day *)
    		enabled := (DATE_TO_DWORD(dat)/86400) MOD (MODE - 10) = 0;
    	20:	(* monday - friday *)
    		enabled := wday <= 5;
    	21:	(* saturday and sunday *)
    		enabled := wday > 5;
    	22: (* workdays only *)
    		enabled := wday <= 5 AND NOT HOLIDAY;
    	23:	(* holidays and weekends *)
    		enabled := wday > 5 OR HOLIDAY;
    	24:	(* holidays only *)
    		enabled := HOLIDAY;
    	25:	(* 1st day of the month *)
    		enabled := DAY_OF_MONTH(dat) = 1;
    	26:	(* last day of month *)
    		enabled := DAY_OF_MONTH(dat + T#1D) = 1;
    	27:	(* 31st of december *)
    		enabled := DAY_OF_MONTH(dat) = 31 AND MONTH_OF_DATE(dat) = 12;
    	28:	(* 1st of january *)
    		enabled := DAY_OF_YEAR(dat) = 1;
    ELSE
    	enabled := FALSE;
    END_CASE

    (* set output if necessary *)
    IF enabled AND NOT Q AND daytime >= START AND run_date <> dat THEN
    	Q := TRUE;
    	activation := tx;
    	run_date := dat;
    ELSIF Q AND tx - activation >= DURATION THEN
    	Q := FALSE;
    END_IF
    last_check := tx;

    (* revision history
    hm 22.2.2007		rev 1.1
    	changed VAR RETAIN PERSISTENT to VAR RETAIN for better compatibility
    	wago lon contollers do not support persisitent

    hm	15.9.2007		rev 1.2
    	replaced Time() with T_PLC_MS for compatibility and performance reasons

    hm	7. oct. 2008	rev 1.3
    	changed function month to month_of_date

    hm	20. oct. 2008	rev 1.4
    	improved performance
    	deleted unnecessary trunc

    hm	22. dec. 2008	rev 1.5
    	make sure timer_2 is executed in the first cycle

    *)
END_FUNCTION_BLOCK

(* ---- TIMER_EXT.st ---- *)
FUNCTION_BLOCK TIMER_EXT
    (*http://www.oscat.de/images/OSCATBuilding/oscat_building100_en.pdf#page=63*)
    (* lösche die millisekunden bei sunrise und sunset *)
    SUN_RISE := DWORD_TO_TOD(TOD_TO_DWORD(SUN_RISE) / 1000 * 1000);
    SUN_SET := DWORD_TO_TOD(TOD_TO_DWORD(SUN_SET) / 1000 * 1000);

    (* measure cycle time tc and make sure this circuitry is not called more then once in 200ms*)
    tx := T_PLC_MS();
    IF NOT init THEN
    	init := TRUE;
    	tl := tx;
    END_IF
    tc := DWORD_TO_TIME(tx - tl);
    IF tc < t#200ms THEN RETURN; END_IF
    tl := tx;

    (* debounce *)
    deb(in := SWITCH, TD := T_DEBOUNCE, PM := TRUE);

    (* read time of day and strip OFF all milliseconds *)
    tdx := DT_TO_TOD(DT_IN);
    wdx := DAY_OF_WEEK(DT_TO_DATE(DT_IN));

    (* automatic output control *)
    IF deb.Q THEN
    	qx := NOT qx;
    	STATUS := 110;
    ELSIF HOLIDAY AND NOT ENABLE_HOLIDAY THEN
    	qx := FALSE;
    ELSIF wdx = 6 AND NOT ENABLE_SATURDAY THEN
    	qx := FALSE;
    ELSIF wdx = 7 AND NOT ENABLE_SUNDAY THEN
    	qx := FALSE;
    ELSIF T_DAY_START > TOD#00:00 AND tdx - T_DAY_START <= tc THEN
    	(* turn ON at specified daytime *)
    	qx := TRUE;
    	STATUS := 111;
    ELSIF T_DAY_STOP > TOD#00:00 AND tdx - T_DAY_STOP <= tc THEN
    	(* turn OFF at specific daytime *)
    	qx := FALSE;
    	STATUS := 112;
    ELSIF T_RISE_START > T#0s AND tdx - SUN_RISE + T_RISE_START <= tc THEN
    	(* turn ON before sunrise *)
    	qx := TRUE;
    	STATUS := 113;
    ELSIF T_RISE_STOP > T#0s AND tdx - SUN_RISE - T_RISE_STOP <= tc THEN
    	(* turn OFF after sunrise *)
    	qx := FALSE;
    	STATUS := 114;
    ELSIF T_SET_START > T#0s AND tdx - SUN_SET + T_SET_START <= tc THEN
    	(* turn ON before sunset *)
    	qx := TRUE;
    	STATUS := 115;
    ELSIF T_SET_STOP > t#0s AND tdx - SUN_SET - T_SET_STOP <= tc THEN
    	(* turn OFF after sunset *)
    	qx := FALSE;
    	STATUS := 116;
    END_IF

    (* mnaual and output control *)
    mx(in := qx, ENA := ENA, ON := ON, OFF := OFF, MAN := MAN);
    Q := mx.Q;

    (* set the STATUS output *)
    IF mx.STATUS > 100 THEN STATUS := mx.STATUS; END_IF

    (*
    hm 	7. oct. 2008	rev 1.0
    	original version

    hm	6. nov. 2008	rev 1.1
    	added default = true for ENA input
    *)
END_FUNCTION_BLOCK

(* ---- TIMER_P4.st ---- *)
FUNCTION_BLOCK TIMER_P4
    (*http://www.oscat.de/images/OSCATBuilding/oscat_building100_en.pdf#page=65*)
    (* for performance reasons we only execute the code at the beginning of a new second *)

    IF RST THEN
    	(* reset all events to last active on 1.1.1970 *)
    	last_execute := DT#1970-1-1-00:00;
    	FOR pos := 0 TO array_max DO
    		IF (PROG[pos].channel >= OFS) AND (PROG[pos].channel < (OFS + 4)) THEN PROG[pos].LAST := last_execute; END_IF
    	END_FOR

    	(* reset all set markers and logic masks *)
    	FOR pos := 0 TO channel_max DO
    		qs[pos] := FALSE;
    	END_FOR

    (* normal operation *)
    ELSIF DTIME <> last_execute THEN
    	(* save the actual second for next execution test *)
    	last_execute := DTIME;

    	(* calculate dt for the start of the day to be used in comparisons *)
    	day_start := DATE_TO_DT(DT_TO_DATE(DTIME));

    	(* set all qn to FALSE *)
    	FOR pos := 0 TO channel_max DO qn[pos] := FALSE; END_FOR

    	(* search the array PROG for timer events *)
    	FOR pos := 0 TO array_max DO
    		event := PROG[pos];
    		channel := event.channel - OFS;
    		IF (event.TYP > 0) AND (channel >= 0) AND (channel <= channel_max) THEN
    			ma[channel] := event.LAND;
    			mo[channel] := event.LOR;
    			CASE event.TYP OF
    				1:	(* daily event *)
    					start := day_start + TOD_TO_TIME(event.start);
    					qn[channel] := DTIME >= start AND DTIME <= start + event.DURATION;

    				2: 	(* event by selected weekdays *)
    					IF (SHR(BYTE#128, DAY_OF_WEEK(DT_TO_DATE(DTIME))) AND event.DAY) > 0 THEN
    						start := day_start + TOD_TO_TIME(event.start);
    						qn[channel] := DTIME >= start AND DTIME <= start + event.DURATION;
    					END_IF

    				3:	(* event every N days *)
    					IF current_day MOD event.DAY = 0 THEN
    						start := day_start + TOD_TO_TIME(event.start);
    						qn[channel] := DTIME >= start AND DTIME <= start + event.DURATION;
    					END_IF

    				10:	(* weekly event exactly once a week the weekday is specified in day, 1= mo *)
    					IF DAY_OF_WEEK(DT_TO_DATE(DTIME)) = BYTE_TO_INT(event.DAY) THEN
    						start := day_start + TOD_TO_TIME(event.start);
    						qn[channel] := DTIME >= start AND DTIME <= start + event.DURATION;
    					END_IF

    				20:	(* monthly event *)
    					IF DAY_OF_MONTH(DT_TO_DATE(DTIME)) = BYTE_TO_INT(event.DAY) THEN
    						start := day_start + TOD_TO_TIME(event.start);
    						qn[channel] := DTIME >= start AND DTIME <= start + event.DURATION;
    					END_IF

    				21:	(* event on last day of month *)
    					IF DT_TO_DATE(DTIME) = MONTH_END(DT_TO_DATE(DTIME)) THEN
    						start := day_start + TOD_TO_TIME(event.start);
    						qn[channel] := DTIME >= start AND DTIME <= start + event.DURATION;
    					END_IF

    				30:	(* yearly event on a specific day specified in day *)
    					IF DAY_OF_YEAR(DT_TO_DATE(DTIME)) = BYTE_TO_INT(event.DAY) THEN
    						start := day_start + TOD_TO_TIME(event.start);
    						qn[channel] := DTIME >= start AND DTIME <= start + event.DURATION;
    					END_IF

    				31:	(* event on last day of year *)
    					IF DT_TO_DATE(DTIME) = YEAR_END(YEAR_OF_DATE(DT_TO_DATE(DTIME))) THEN
    						start := day_start + TOD_TO_TIME(event.start);
    						qn[channel] := DTIME >= start AND DTIME <= start + event.DURATION;
    					END_IF

    				40:	(* event on leap days *)
    					IF LEAP_DAY(DT_TO_DATE(DTIME)) THEN
    						start := day_start + TOD_TO_TIME(event.start);
    						qn[channel] := DTIME >= start AND DTIME <= start + event.DURATION;
    					END_IF

    				41: (* event on holidays *)
    					IF HOLY THEN
    						start := day_start + TOD_TO_TIME(event.start);
    						qn[channel] := DTIME >= start AND DTIME <= start + event.DURATION;
    					END_IF

    				42: (* event on holidays and weekends *)
    					IF (HOLY OR (DAY_OF_WEEK(DT_TO_DATE(DTIME)) = 6) OR (DAY_OF_WEEK(DT_TO_DATE(DTIME)) = 7)) THEN
    						start := day_start + TOD_TO_TIME(event.start);
    						qn[channel] := DTIME >= start AND DTIME <= start + event.DURATION;
    					END_IF

    				43:	(* event on workdays mo-FR and no holiday *)
    					IF DAY_OF_WEEK(DT_TO_DATE(DTIME)) < 6 THEN
    						start := day_start + TOD_TO_TIME(event.start);
    						qn[channel] := DTIME >= start AND DTIME <= start + event.DURATION;
    					END_IF

    				50: (* event after reference time *)
    					CASE PROG[pos].DAY OF
    						0:	tx := TREF_0;
    						1:	tx := TREF_1;
    					ELSE
    						tx := TOD#00:00;
    					END_CASE
    					start := day_start + TOD_TO_TIME(tx) + TOD_TO_TIME(event.start);
    					qn[channel] := DTIME >= start AND DTIME <= start + event.DURATION;

    				51:	(* event before reference time *)
    					CASE PROG[pos].DAY OF
    						0:	tx := TREF_0;
    						1:	tx := TREF_1;
    					ELSE
    						tx := TOD#00:00;
    					END_CASE
    					start := day_start + TOD_TO_TIME(tx) - TOD_TO_TIME(event.start);
    					qn[channel] := DTIME >= start AND DTIME <= start + event.DURATION;

    				52 : (* set output at specific time + offset  *)
    					CASE PROG[pos].DAY OF
    						0:	tx := TREF_0;
    						1:	tx := TREF_1;
    					ELSE
    						tx := TOD#00:00;
    					END_CASE
    					start := day_start + TOD_TO_TIME(tx) + TOD_TO_TIME(event.start);
    					IF DTIME >= start AND day_start > event.LAST THEN
    						qs[channel] := TRUE;
    						PROG[pos].LAST := day_start;
    					END_IF

    				53 : (* reset output at specific time + offset *)
    					CASE PROG[pos].DAY OF
    						0:	tx := TREF_0;
    						1:	tx := TREF_1;
    					ELSE
    						tx := TOD#00:00;
    					END_CASE
    					start := day_start + TOD_TO_TIME(tx) + TOD_TO_TIME(event.start);
    					IF DTIME >= start AND day_start > event.LAST THEN
    						qs[channel] := FALSE;
    						PROG[pos].LAST := day_start;
    					END_IF

    				54 : (* set output at specific time - offset  *)
    					CASE PROG[pos].DAY OF
    						0:	tx := TREF_0;
    						1:	tx := TREF_1;
    					ELSE
    						tx := TOD#00:00;
    					END_CASE
    					start := day_start + TOD_TO_TIME(tx) - TOD_TO_TIME(event.start);
    					IF DTIME >= start AND day_start > event.LAST THEN
    						qs[channel] := TRUE;
    						PROG[pos].LAST := day_start;
    					END_IF

    				55 : (* reset output at specific time - offset *)
    					CASE PROG[pos].DAY OF
    						0:	tx := TREF_0;
    						1:	tx := TREF_1;
    					ELSE
    						tx := TOD#00:00;
    					END_CASE
    					start := day_start + TOD_TO_TIME(tx) - TOD_TO_TIME(event.start);
    					IF DTIME >= start AND day_start > event.LAST THEN
    						qs[channel] := FALSE;
    						PROG[pos].LAST := day_start;
    					END_IF
    			END_CASE
    		END_IF
    	END_FOR
    END_IF

    (* prepare the logical input mask *)
    mask := 255;
    mask.0 := L0;
    mask.1 := L1;
    mask.2 := L2;
    mask.3 := L3;

    (* set the outputs *)
    Q0 := ENQ AND ((qn[0] OR qs[0]) AND ((ma[0] AND mask) = ma[0]) OR ((mo[0] AND mask) > 0) OR (MAN AND MI.0));
    Q1 := ENQ AND ((qn[1] OR qs[1]) AND ((ma[1] AND mask) = ma[1]) OR ((mo[1] AND mask) > 1) OR (MAN AND MI.1));
    Q2 := ENQ AND ((qn[2] OR qs[2]) AND ((ma[2] AND mask) = ma[2]) OR ((mo[2] AND mask) > 2) OR (MAN AND MI.2));
    Q3 := ENQ AND ((qn[3] OR qs[3]) AND ((ma[3] AND mask) = ma[3]) OR ((mo[3] AND mask) > 3) OR (MAN AND MI.3));

    (* set STATUS *)
    IF NOT ENQ THEN
    	STATUS := 100;
    ELSIF MAN THEN
    	STATUS := 101;
    ELSE
    	STATUS := 102;
    END_IF

    (* revision history
    hm	17. jun 2008	rev 1.0
    	original version

    hm	9. oct. 2008	rev 1.1
    	changed function year to year_of_date
    	changed function weekday to day_of_week
    	changed structure of program to be more efficient
    	changed input DIS to ENQ

    hm	18. oct. 2008	rev 1.2
    	changed type of input OFS from int to byte
    	added typecasts to avoid warnings

    hm	28. feb. 2009	rev 1.3
    	array was not correctly initialized

    hm	26. jan 2011	rev 1.4
    	changed code to allow events over midnight
    *)

END_FUNCTION_BLOCK

(* ---- oscatBuild.var ---- *)
VAR CONSTANT
END_VAR
